FUNCTION "FC_1" : Void
{ S7_Optimized_Access := 'TRUE' }
VERSION : 0.1
   VAR_INPUT
      input : Real;
   END_VAR

   VAR_OUTPUT
      output : Real;
   END_VAR


BEGIN
	#output := #input * 15.0;

END_FUNCTION

